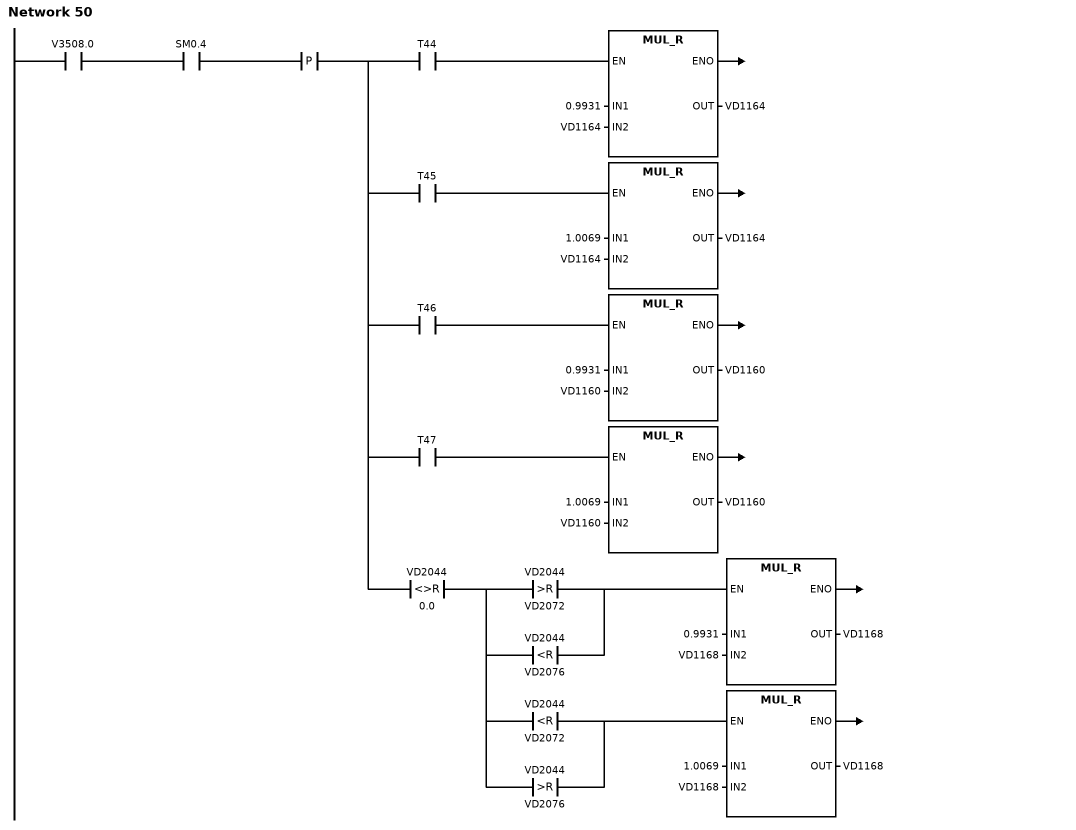
[picture p24: SBR0 networks 50-50]
Network 50
LD     V3508.0
A      SM0.4
EU
LPS
A      T44
*R     0.9931, VD1164
LRD
A      T45
*R     1.0069, VD1164
LRD
A      T46
*R     0.9931, VD1160
LRD
A      T47
*R     1.0069, VD1160
LPP
AR<>   VD2044, 0.0
LPS
LDR>   VD2044, VD2072
OR<    VD2044, VD2076
ALD
*R     0.9931, VD1168
LPP
LDR<   VD2044, VD2072
OR>    VD2044, VD2076
ALD
*R     1.0069, VD1168
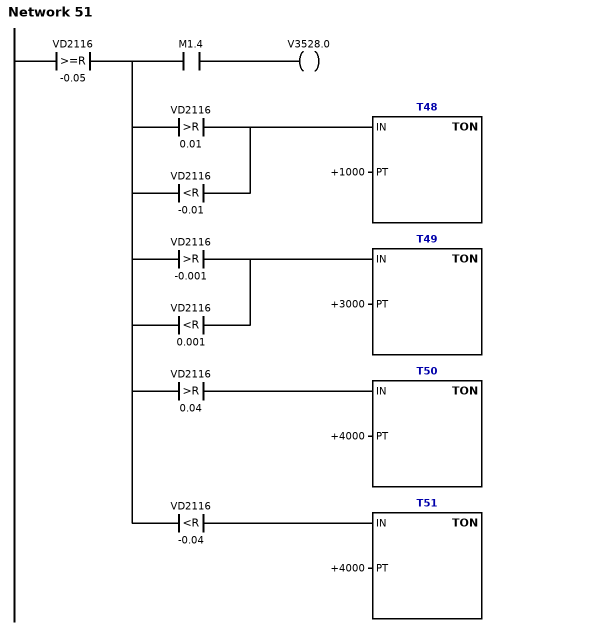
Network 51
LDR>=  VD2116, -0.05
LPS
A      M1.4
=      V3528.0
LRD
LDR>   VD2116, 0.01
OR<    VD2116, -0.01
ALD
TON    T48, +1000
LRD
LDR>   VD2116, -0.001
OR<    VD2116, 0.001
ALD
TON    T49, +3000
LPP
LPS
AR>    VD2116, 0.04
TON    T50, +4000
LPP
AR<    VD2116, -0.04
TON    T51, +4000
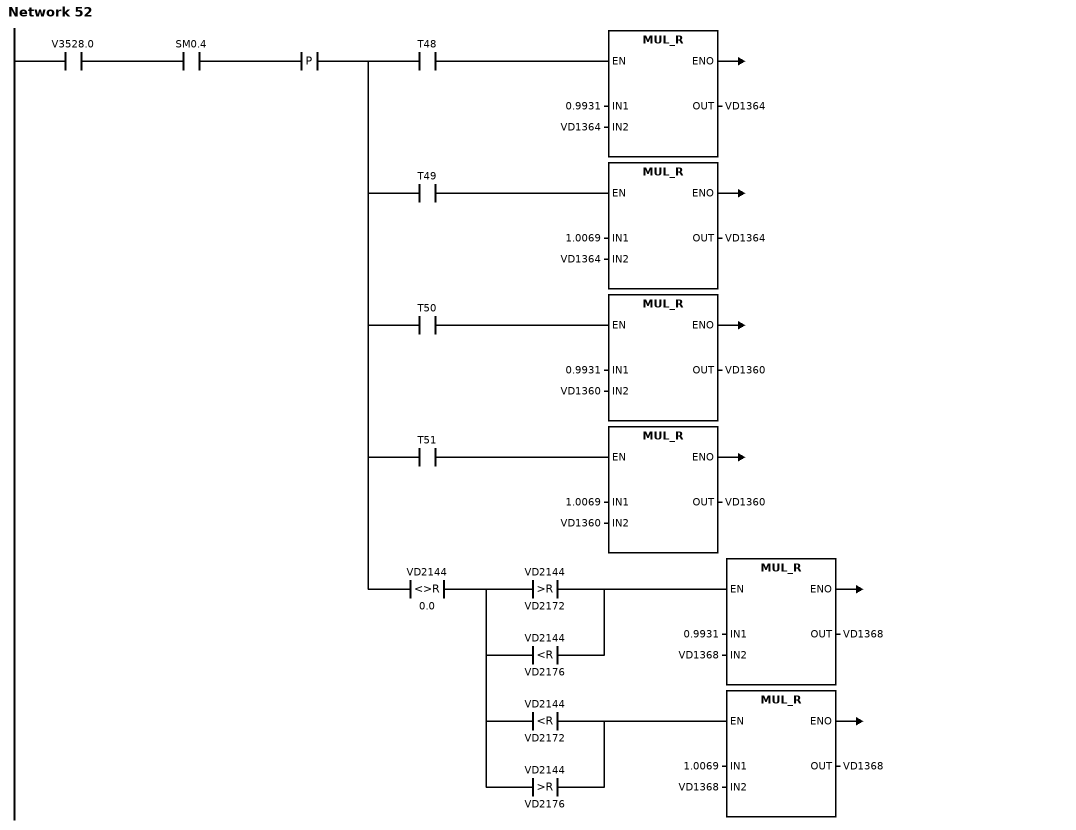
Network 52
LD     V3528.0
A      SM0.4
EU
LPS
A      T48
*R     0.9931, VD1364
LRD
A      T49
*R     1.0069, VD1364
LRD
A      T50
*R     0.9931, VD1360
LRD
A      T51
*R     1.0069, VD1360
LPP
AR<>   VD2144, 0.0
LPS
LDR>   VD2144, VD2172
OR<    VD2144, VD2176
ALD
*R     0.9931, VD1368
LPP
LDR<   VD2144, VD2172
OR>    VD2144, VD2176
ALD
*R     1.0069, VD1368
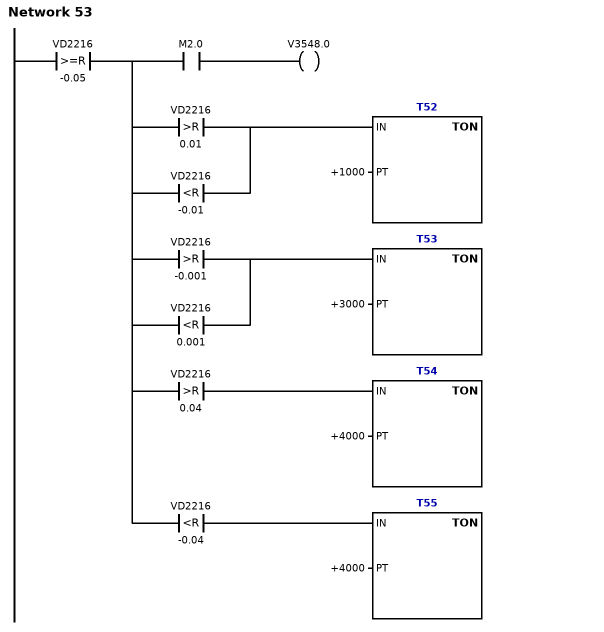
Network 53
LDR>=  VD2216, -0.05
LPS
A      M2.0
=      V3548.0
LRD
LDR>   VD2216, 0.01
OR<    VD2216, -0.01
ALD
TON    T52, +1000
LRD
LDR>   VD2216, -0.001
OR<    VD2216, 0.001
ALD
TON    T53, +3000
LPP
LPS
AR>    VD2216, 0.04
TON    T54, +4000
LPP
AR<    VD2216, -0.04
TON    T55, +4000
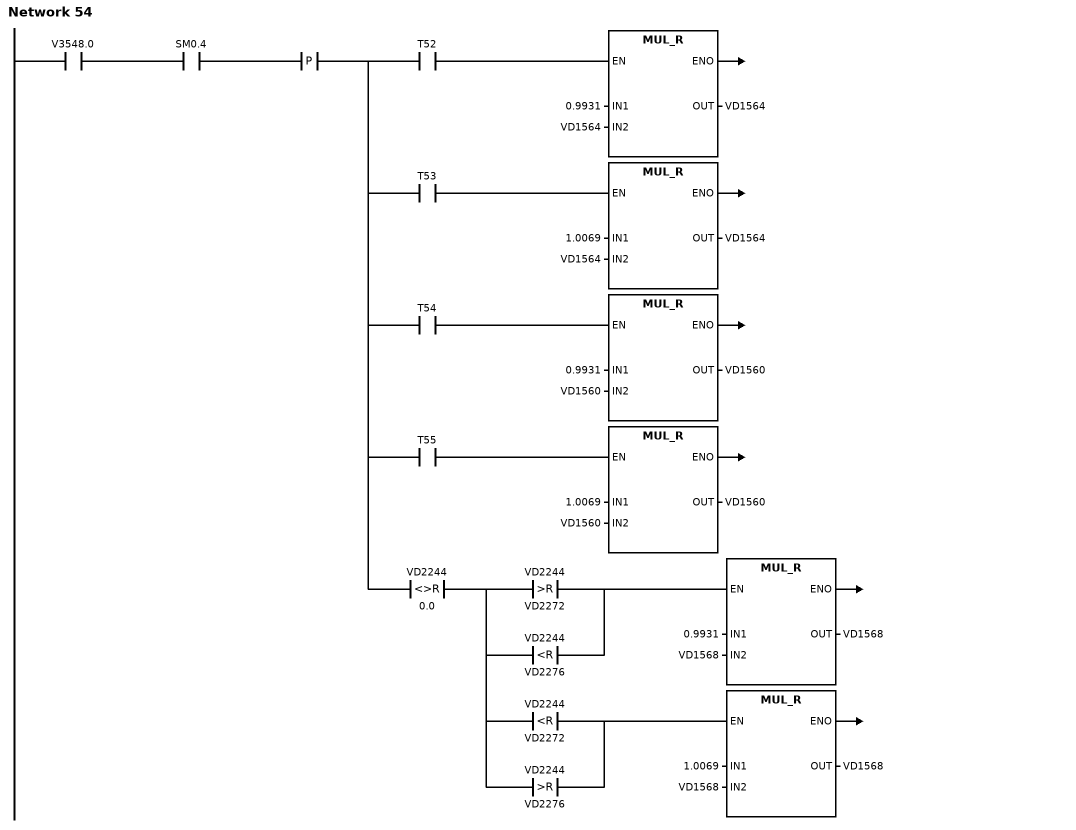
Network 54
LD     V3548.0
A      SM0.4
EU
LPS
A      T52
*R     0.9931, VD1564
LRD
A      T53
*R     1.0069, VD1564
LRD
A      T54
*R     0.9931, VD1560
LRD
A      T55
*R     1.0069, VD1560
LPP
AR<>   VD2244, 0.0
LPS
LDR>   VD2244, VD2272
OR<    VD2244, VD2276
ALD
*R     0.9931, VD1568
LPP
LDR<   VD2244, VD2272
OR>    VD2244, VD2276
ALD
*R     1.0069, VD1568
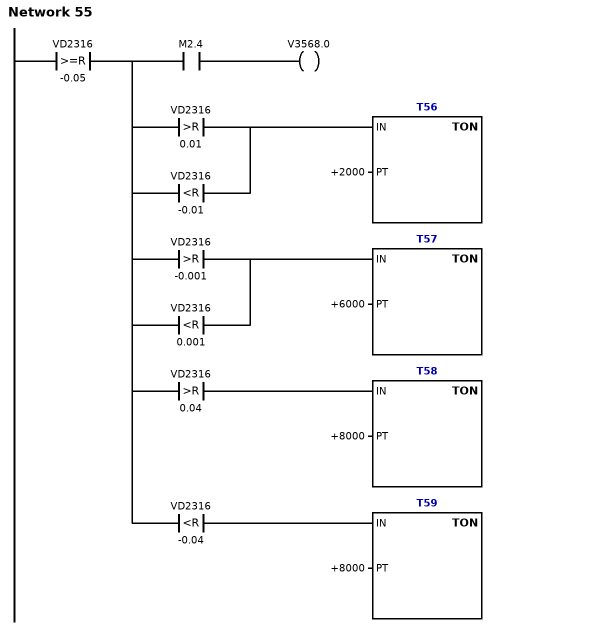
Network 55
LDR>=  VD2316, -0.05
LPS
A      M2.4
=      V3568.0
LRD
LDR>   VD2316, 0.01
OR<    VD2316, -0.01
ALD
TON    T56, +2000
LRD
LDR>   VD2316, -0.001
OR<    VD2316, 0.001
ALD
TON    T57, +6000
LPP
LPS
AR>    VD2316, 0.04
TON    T58, +8000
LPP
AR<    VD2316, -0.04
TON    T59, +8000
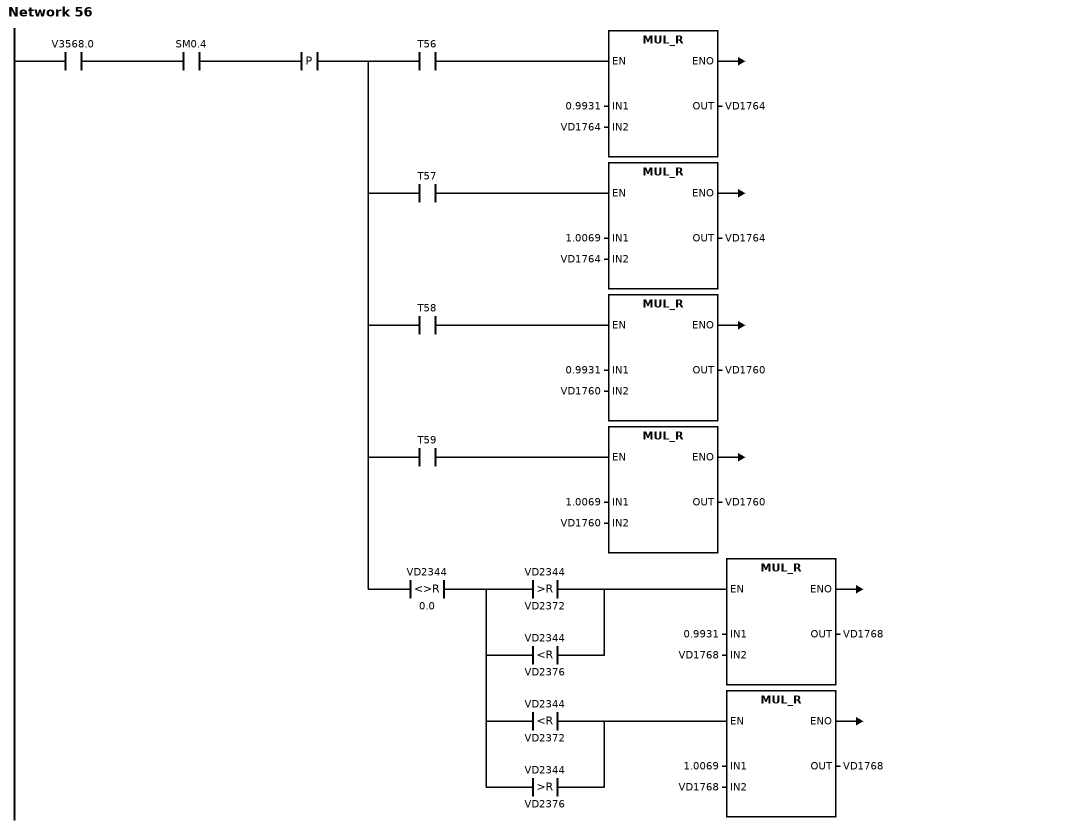
Network 56
LD     V3568.0
A      SM0.4
EU
LPS
A      T56
*R     0.9931, VD1764
LRD
A      T57
*R     1.0069, VD1764
LRD
A      T58
*R     0.9931, VD1760
LRD
A      T59
*R     1.0069, VD1760
LPP
AR<>   VD2344, 0.0
LPS
LDR>   VD2344, VD2372
OR<    VD2344, VD2376
ALD
*R     0.9931, VD1768
LPP
LDR<   VD2344, VD2372
OR>    VD2344, VD2376
ALD
*R     1.0069, VD1768
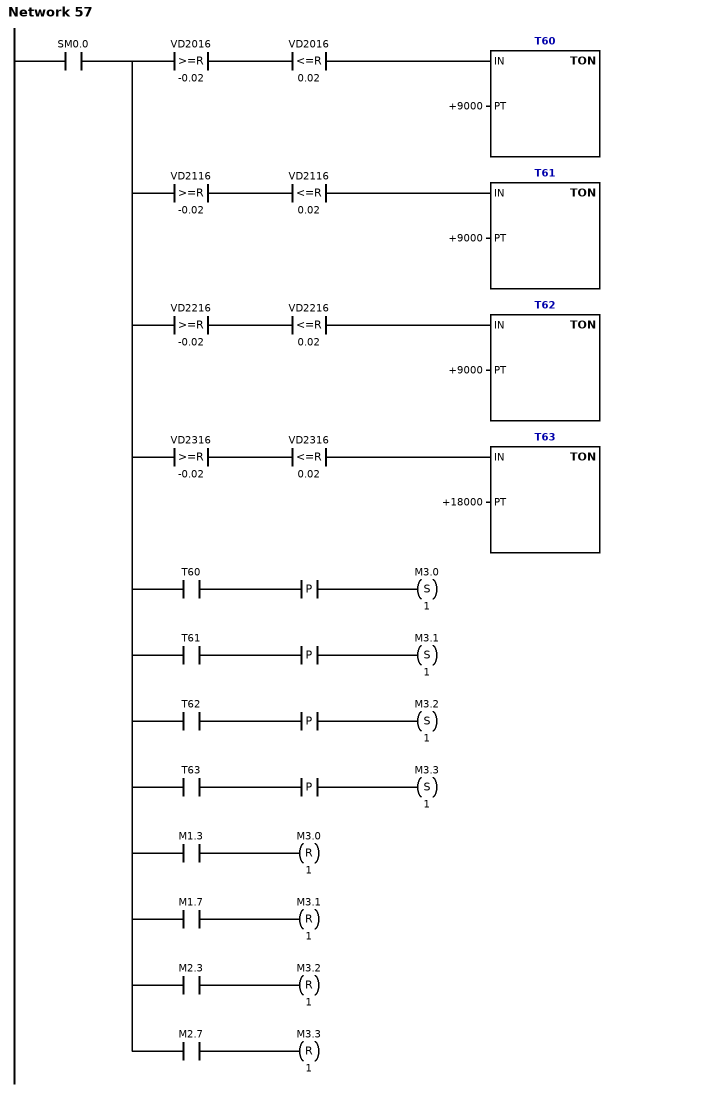
Network 57
LD     SM0.0
LPS
AR>=   VD2016, -0.02
AR<=   VD2016, 0.02
TON    T60, +9000
LRD
AR>=   VD2116, -0.02
AR<=   VD2116, 0.02
TON    T61, +9000
LRD
AR>=   VD2216, -0.02
AR<=   VD2216, 0.02
TON    T62, +9000
LRD
AR>=   VD2316, -0.02
AR<=   VD2316, 0.02
TON    T63, +18000
LRD
A      T60
EU
S      M3.0, 1
LRD
A      T61
EU
S      M3.1, 1
LRD
A      T62
EU
S      M3.2, 1
LRD
A      T63
EU
S      M3.3, 1
LRD
A      M1.3
R      M3.0, 1
LRD
A      M1.7
R      M3.1, 1
LRD
A      M2.3
R      M3.2, 1
LPP
A      M2.7
R      M3.3, 1
END_SUBROUTINE_BLOCK

// SBR1: protected block, not included

// SBR2: protected block, not included

// SBR3: protected block, not included

// SBR5: protected block, not included

// SBR6: protected block, not included

DATA_BLOCK_TAB 用户定义1
BEGIN
VD1050   180
VD1054   15
VD1058   1900
VD1062   300
VD1130   5.0
VD1142   1.0
VD1134   1.15
VD1138   0.0002
VD1330   5.0
VD1342   1.0
VD1334   1.15
VD1338   0.0002
VD1530   5.0
VD1542   1.0
VD1534   1.15
VD1538   0.0002
VD1730   5.0
VD1742   1.0
VD1734   50.0
VD1738   0.002
END_DATA_BLOCK_TAB
